INTERFACE I_Disposable

METHOD Dispose
VAR_INPUT
END_VAR
END_METHOD

END_INTERFACE

(* stored: Version 1.1.0.1, ProductVersion 3.1.4024.12
   Itf I_Disposable: Id {2f7ea90b-3a9c-44d0-a95f-bfbb63cc1a95}
   Method Dispose: Id {5a3a9860-dfbf-472d-bf18-0155c1e57262} *)
